{attribute 'qualified_only'}
{attribute 'strict'}
TYPE eBeltObject :
(
	EMPTY := 0,
	GATO := 1,
	PERRO := 2,
	MAGIC := 3
);
END_TYPE

(* stored: Version 1.1.0.1, ProductVersion 3.1.4024.10
   DUT eBeltObject: Id {2bbc16ef-bc8b-453a-9b00-8cdd4b4915b7} *)
